FUNCTION_BLOCK FB_FireShowModeCommand IMPLEMENTS I_Command
VAR
	refFlameCannon : REFERENCE TO FB_FlameCannon;
END_VAR

METHOD Execute
IF (__ISVALIDREF(THIS^.refFlameCannon)) THEN
	THIS^.refFlameCannon.On();
	THIS^.refFlameCannon.SetLevel(25.50);
END_IF
END_METHOD

METHOD FB_init : BOOL
VAR_INPUT
	bInitRetains 	: BOOL; // if TRUE, the retain variables are initialized (warm start / cold start)
	bInCopyCode 	: BOOL;  // if TRUE, the instance afterwards gets moved into the copy code (online change)
	refFlameCannon 	: REFERENCE TO FB_FlameCannon;
END_VAR
IF (__ISVALIDREF(refFlameCannon)) THEN
	THIS^.refFlameCannon REF= refFlameCannon;
ELSE
	THIS^.refFlameCannon REF= 0;
END_IF
END_METHOD

END_FUNCTION_BLOCK

(* stored: Version 1.1.0.1, ProductVersion 3.1.4022.18
   POU FB_FireShowModeCommand: Id {3a8e07f3-a49c-4672-bc9c-28982628a694}, SpecialFunc None
   Method Execute: Id {5c65ece6-6212-47d0-a3f4-f573b03597e9}
   Method FB_init: Id {08a5122f-d44a-4309-9dac-b4a15da6e11e} *)
